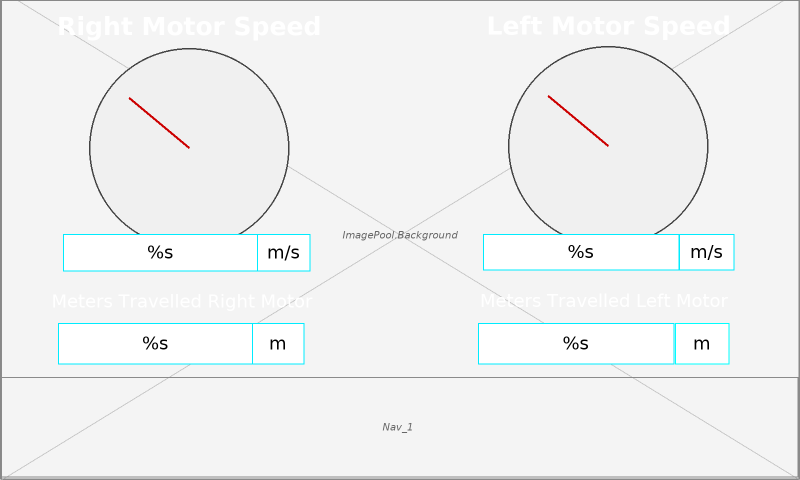
VISUALIZATION Charge_Velocity_Distance  // 800x480
    Image (1,-10 799x490), image: ImagePool.Background
    Meter180 (14,48 350x200), value: MAIN.RightVelocityValue, style: Meter-Meter180-Green, scale format: %.1f, scale 0..0.7
        p518627256: m/s
    Meter180 (433,46 350x200), value: MAIN.LeftVelocityValue, style: Meter-Meter180-Green, scale format: %.1f, scale 0..0.7
        p518627256: m/s
    RoundedRectangle (57,10 265x32), "Right Motor Speed"
    RoundedRectangle (478,10 262x31), "Left Motor Speed"
    Textfield (63,234 195x37), "%s", text variable: MAIN.RightVelocityValue
    Textfield (483,234 196x36), "%s", text variable: MAIN.LeftVelocityValue
    Rectangle (257,234 53x37), "m/s"
    BarDisplayImage (823,379 336x111), style: BarDisplayImage-Yellow, scale format: %.1f, scale 0..100
    RoundedRectangle (463,281 282x40), "Meters Travelled Left Motor"
    Textfield (58,323 195x41), "%s", text variable: Meters_Travelled.r_meters_travelled
    Rectangle (252,323 52x41), "m"
    RoundedRectangle (41,282 282x39), "Meters Travelled Right Motor"
    Textfield (478,323 196x41), "%s", text variable: Meters_Travelled.l_meters_travelled
    Rectangle (675,323 54x41), "m"
    Rectangle (679,234 55x36), "m/s"
    Frame (-2,377 800x100)
        shows Nav_1()
END_VISUALIZATION

(* stored: Version 1.1.0.1, ProductVersion 3.1.4024.12
   Visu Charge_Velocity_Distance: Id {b9a73025-959e-4dfa-adb8-eaaf5032d426} *)
